// TIA Portal V20 export
DATA_BLOCK "ComErr"   // DB363
{ S7_Optimized_Access := 'FALSE' }
// stored: AutoNumber false
   VAR
      Plc : "TypeHeaderPlc";   // Header Plc
      Pc : "TypeHeaderPcGld";   // Header Pc
      Err : Array[2000..2599] of Bool;
   END_VAR
BEGIN
END_DATA_BLOCK
